FUNCTION_BLOCK ResetARM (* Basic Function Block Type *)
  (* Standard: 61499-2 *)
  (* Version 0.0, 2/12/2018, Sandeep Patil, nxtControl GmbH, Template *)
  PACKAGE Main;
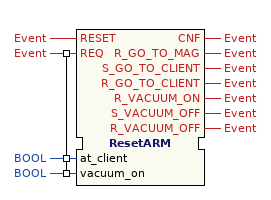
  EVENT_INPUT
    RESET; (* Initialization Request *)
    REQ WITH at_client, vacuum_on;
  END_EVENT
  EVENT_OUTPUT
    CNF; (* Initialization Confirm *)
    R_GO_TO_MAG; (* Execution Confirmation *)
    S_GO_TO_CLIENT; (* Initialization Confirm *)
    R_GO_TO_CLIENT; (* Execution Confirmation *)
    R_VACUUM_ON; (* Execution Confirmation *)
    S_VACUUM_OFF; (* Initialization Confirm *)
    R_VACUUM_OFF; (* Execution Confirmation *)
  END_EVENT
  VAR_INPUT
    at_client : BOOL;
    vacuum_on : BOOL;
  END_VAR
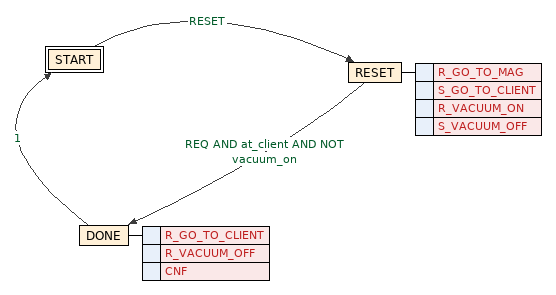
  EC_STATES
    START; (* Initial State *)
    RESET : -> R_GO_TO_MAG, -> S_GO_TO_CLIENT, -> R_VACUUM_ON, -> S_VACUUM_OFF; (* Normal execution *)
    DONE : -> R_GO_TO_CLIENT, -> R_VACUUM_OFF, -> CNF;
  END_STATES
  EC_TRANSITIONS
    START TO RESET := RESET;
    RESET TO DONE := REQ AND at_client AND NOT vacuum_on;
    DONE TO START := 1;
  END_TRANSITIONS
END_FUNCTION_BLOCK
